FUNCTION_BLOCK AUI_MUX_8 (* Event multiplexer with AUI adapter output instead of plain EO+K (generic FB) *)
  (* Standard: 61499-1 Annex A; Description: Copyright (c) 2017, 2025 fortiss GmbH, HR Agrartechnik GmbH This program and the accompanying materials are made available under the terms of the Eclipse Public License 2.0 which is available at https://www.eclipse.org/legal/epl-2.0/ SPDX-License-Identifier: EPL-2.0 *)
  (* Version 3.0, 2025-04-14, Patrick Aigner, changed package *)
  (* Version 1.1, 2025-02-16, Franz Höpfinger, HR Agrartechnik GmbH, Copy E_DEMUX8 and made E_MUX8 *)
  (* Version 1.0, 2017-09-22, Alois Zoitl, fortiss GmbH, initial API and implementation and/or initial documentation *)
  PACKAGE adapter::events::unidirectional;
  {SET_ATTRIBUTE(eclipse4diac::core::GenericClassName, 'GEN_AUI_MUX')}
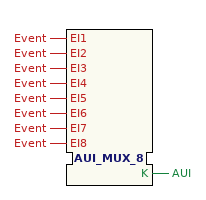
  EVENT_INPUT
    EI1; (* Event to multiplex, K=0 *)
    EI2; (* Event to multiplex, K=1 *)
    EI3; (* Event to multiplex, K=2 *)
    EI4; (* Event to multiplex, K=3 *)
    EI5; (* Event to multiplex, K=4 *)
    EI6; (* Event to multiplex, K=5 *)
    EI7; (* Event to multiplex, K=6 *)
    EI8; (* Event to multiplex, K=7 *)
  END_EVENT
  PLUGS
    K : adapter::types::unidirectional::AUI; (* Event index *)
  END_PLUGS
END_FUNCTION_BLOCK
